// TIA Portal V17 export
// export: Created 2022-07-28T18:03:17.7297808Z, ExportSetting None, DisplayName Totally Integrated Automation Portal, DisplayVersion V17, DisplayName TIA Portal Openness, DisplayVersion V17, DisplayName TIA Portal Teamcenter Gateway, DisplayVersion V17, DisplayName TIA Portal Version Control Interface, DisplayVersion V17, DisplayName TIA Portal Test Suite Advanced, DisplayVersion V17, DisplayName SINAMICS Startdrive Advanced, DisplayVersion V17, DisplayName SINAMICS DCC, DisplayVersion V17, DisplayName SINAMICS Startdrive G130, G150, S120, S150, SINAMICS MV, S210, DisplayVersion V17, DisplayName SINAMICS Startdrive G110M, G120, G120C, G120D, G120P, G115D, DisplayVersion V17, DisplayName STEP 7 Professional, DisplayVersion V17, DisplayName SIMATIC Energy Suite, DisplayVersion V17, DisplayName STEP 7 CFC, DisplayVersion V17, DisplayName STEP 7 Safety, DisplayVersion V17, DisplayName WinCC Advanced / Unified PC, DisplayVersion V17, DisplayName SIMATIC Visualization Architect, DisplayVersion V17
TYPE "Lib_UDT_PLC"
   STRUCT
      ID : Int;   // Унікальний ідентифікатор
      CMD : Int;   // Команди з HMI
      PLS { S7_SetPoint := 'True'} : "Lib_PLC_PLS";   // бітові міандри
      CycleInfo { S7_SetPoint := 'True'} : "Lib_PLC_CycleInfo";
      CMDPRG : UInt;   // Команди з програмного керування (побітові)
      PRM1 : UInt;   // дискретні параметри
      PRM2 : UInt;   // дискретні параметри
      Alarm2 : Int;   // біти алармів
      STEP1 : Int;   // крок основної програми
      T_STEP1 : Int;   // час кроку основної програми обробки, в (с)
      Message : UDInt;   // для формування повідомлень, може бути як бітовим (32 повідомлення), так і числовим (за номером); передбачається, що повідомлення буде скидуватися в 0 автоматично через певний час (не менш ніж 2 інтервали опитування з HMI)
      NumberDI : Int;   // кількість наявних каналів DI
      NumberDO : Int;   // кількість наявних каналів DO
      NumberAI : Int;   // кількість наявних каналів AI
      NumberAO : Int;   // кількість наявних каналів AO
      NOW : Array[0..3] of Int;   // плинний час астрономічний час в BCD форматі: NOW[0] seconds,-- (16#ss,--) NOW[1] hour, minute (16#hhmm) NOW[2] month, day (16#mmdd) NOW[3] year (16#yyyy)
      ShiftParam : Array[0..3] of Int;   // Години передачі змін (максимум 3 зміни): SHIFT[0] – кількість змін SHIFT[1] – передача 1-ї зміни (BCD 16#hhmm) SHIFT[2] – передача 2-ї зміни (BCD 16#hhmm) SHIFT[3] – передача 3-ї зміни (BCD 16#hhmm)
      ShiftActiveNumber : Int;   // номер активної зміни
      TSK_LTIME : LTime;   // плинний (останній) час задачі в мілісекундах
      TSK_MAXTIME : LTime;   // максимальний час задачі в мілісекундах
      TSK_MINTIME : LTime;   // максимальний час задачі в мілісекундах
      TaskTime : "Lib_PLC_TaskTime";   // RT_INFO
      TIME_TCK : Struct
         cyclic_sec_R { ExternalVisible := 'False'; ExternalWritable := 'False'} : Real;   // !!_ЧАС ЦИКЛУ_!!!
         cyclic_ms { ExternalVisible := 'False'; ExternalWritable := 'False'} : Int;   // msec, Плинне/поточне значення часу виконання циклу циклу OB1
         cyclic_sec_LR { ExternalVisible := 'False'; ExternalWritable := 'False'} : LReal;   // sec, Плинне/поточне значення часу виконання циклу циклу OB1
         FirstScanTime { ExternalVisible := 'False'; ExternalWritable := 'False'} : Date_And_Time;   // Дата/час "FirstScan"
         PrevScanTime { ExternalVisible := 'False'; ExternalWritable := 'False'} : Date_And_Time;   // Дата/час попередньго виклику OB1
         NowTime { ExternalWritable := 'False'} : Date_And_Time;   // Дата/час поточні
         Time1cycle_r : LReal;   // загальний час з початку 1-го циклу контролера (в секундах)
         Time1cycle_di : UDInt;   // загальний час з початку 1-го циклу контролера (в секундах)
         Time1cycle_DINT : UDInt;   // sec, Час від "FirstScan"
         TimeTotalPLC : UDInt;   // загальний час роботи ПЛК з моменту пуску (в хвилинах)
      END_STRUCT;
      TaskTime_RUNTIME : Struct   // RUNTIME
         Live : LReal;   // sec, Плинне/поточне значення часу виконання блоку
         TIME_TCK_s : LReal;   // sec, Час від першого циклу
      END_STRUCT;
      MEM_RUNTIME { S7_SetPoint := 'True'} : LReal;
      HMI : Struct
         State : UDInt;   // повторює STA, який був на початку виклику функції
         Alarm : UDInt;   // повторює ALM1, який був на початку виклику функції
         "Counter" : "Lib_PLC_AlarmCounter";
      END_STRUCT;
   END_STRUCT;
END_TYPE
